// TIA Portal project "Paso a paso S7-1200 cambio giro bien en ambos sentidos intento completo final" (V16)

(* hardware
DEVICE "S7-1200 station_1"  S7-1200 Station
   slot 0: "Rack_0"  S7-1200 Rack  Rack  V1.0
   slot 1: "PLC_1"  CPU 1214C DC/DC/DC  6ES7 214-1AG31-0XB0  V3.0
*)

// ===== PLC "PLC_1"  CPU 1214C DC/DC/DC =====

VAR_GLOBAL   // PLC tag table "Tabla de variables estándar"
   "Marcha" AT %I0.1 : Bool;
   "Paro" AT %I0.2 : Bool;
   "IN1" AT %Q0.0 : Bool;
   "IN2" AT %Q0.1 : Bool;
   "IN3" AT %Q0.2 : Bool;
   "IN4" AT %Q0.3 : Bool;
   "marca_marcha" AT %M0.0 : Bool;
   "flanco_marcha" AT %M0.1 : Bool;
   "tiempo_trans" AT %MD2 : DInt;
   "marca_reinicio_temp" AT %M0.2 : Bool;
   "tiempo_actual" AT %MD6 : DInt;
   "marca1" AT %MD10 : Real;
   "marca2" AT %MD14 : Real;
   "Emergencia" AT %I0.3 : Bool;
   "Aumento" AT %I0.4 : Bool;
   "Freno" AT %I0.5 : Bool;
   "Conmutador cambio giro" AT %I0.6 : Bool;
   "flanco_aumento" AT %M0.3 : Bool;
   "flanco_freno" AT %M0.4 : Bool;
   "marca_bloqueo_aume_fre" AT %M0.5 : Bool;
   "flanco_paro" AT %M0.6 : Bool;
   "bloqueo_paro" AT %M0.7 : Bool;
   "marca3" AT %MD18 : Real;
   "tiempo_paro" AT %MW26 : Int;
   "marca_paro_a_0" AT %M1.0 : Bool;
   "marca_marcha2" AT %M1.1 : Bool;
   "flanco1" AT %M1.4 : Bool;
   "Inversor de giro" AT %I0.7 : Bool;
   "marca5" AT %M1.2 : Bool;
   "reinicio_counter" AT %M1.3 : Bool;
   "giro_izquierda" AT %M1.5 : Bool;
   "giro_derecha" AT %M1.6 : Bool;
   "estado_derecha" AT %M1.7 : Bool;
   "estado_izquierda" AT %M22.0 : Bool;
   "cambio a izq" AT %M22.1 : Bool;
   "tiempo_cambio" AT %MW30 : Int;
   "marca6" AT %M22.2 : Bool;
   "bloqueo_final" AT %M22.3 : Bool;
   "marca4" AT %MD32 : Real;
   "paro_bloqueo" AT %M22.4 : Bool;
   "tiempo para paro" AT %MW36 : Int;
END_VAR

// folder: System blocks/Program resources

DATA_BLOCK "IEC_Timer_0_DB"   // DB1
{ S7_Optimized_Access := 'TRUE' }
AUTHOR : Simatic
FAMILY : IEC
NAME : IEC_TMR
VERSION : 1.0
// stored: InstanceOfName IEC_TIMER
"IEC_TIMER"
BEGIN
END_DATA_BLOCK

DATA_BLOCK "IEC_Timer_0_DB_1"   // DB2
{ S7_Optimized_Access := 'TRUE' }
AUTHOR : Simatic
FAMILY : IEC
NAME : IEC_TMR
VERSION : 1.0
// stored: InstanceOfName IEC_TIMER
"IEC_TIMER"
BEGIN
END_DATA_BLOCK

DATA_BLOCK "IEC_Counter_0_DB"   // DB3
{ S7_Optimized_Access := 'TRUE' }
AUTHOR : Simatic
FAMILY : IEC
NAME : CNTR
VERSION : 1.0
// stored: InstanceOfName IEC_COUNTER
"IEC_COUNTER"
BEGIN
END_DATA_BLOCK

DATA_BLOCK "IEC_Timer_0_DB_2"   // DB4
{ S7_Optimized_Access := 'TRUE' }
AUTHOR : Simatic
FAMILY : IEC
NAME : IEC_TMR
VERSION : 1.0
// stored: InstanceOfName IEC_TIMER
"IEC_TIMER"
BEGIN
END_DATA_BLOCK

DATA_BLOCK "IEC_Counter_0_DB_1"   // DB5
{ S7_Optimized_Access := 'TRUE' }
AUTHOR : Simatic
FAMILY : IEC
NAME : CNTR
VERSION : 1.0
// stored: InstanceOfName IEC_COUNTER
"IEC_COUNTER"
BEGIN
END_DATA_BLOCK

DATA_BLOCK "IEC_Timer_0_DB_3"   // DB6
{ S7_Optimized_Access := 'TRUE' }
AUTHOR : Simatic
FAMILY : IEC
NAME : IEC_TMR
VERSION : 1.0
// stored: InstanceOfName IEC_TIMER
"IEC_TIMER"
BEGIN
END_DATA_BLOCK

// folder: (top level)

ORGANIZATION_BLOCK "Main"   // OB1, LAD, ProgramCycle
TITLE = "Main Program Sweep (Cycle)"
{ S7_Optimized_Access := 'TRUE' }
VERSION : 0.1
   VAR_TEMP   // added for the SCL form of the ladder/FBD networks
      _w1 : Bool;
      _w2 : Bool;
      _w3 : Bool;
      _w4 : Bool;
      _w5 : Bool;
   END_VAR
BEGIN

REGION Network 1: Marcha
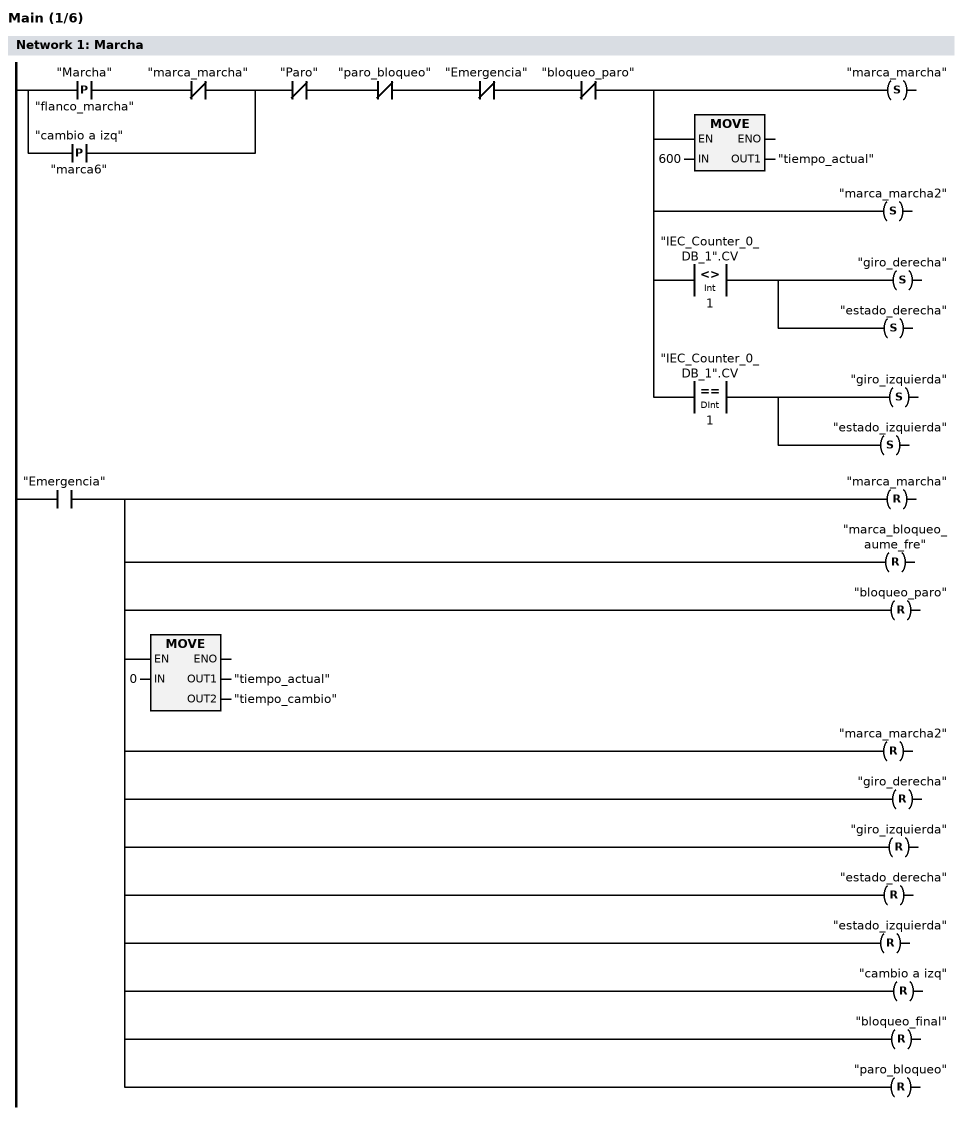
   RUNG wire#powerrail
      P_Contact(operand := "Marcha", bit := "flanco_marcha")
      I_Contact( "marca_marcha" )
      wire#w1
      I_Contact( "Paro" )
      I_Contact( "paro_bloqueo" )
      I_Contact( "Emergencia" )
      I_Contact( "bloqueo_paro" )
      wire#w2
      S_Coil( "marca_marcha" )
   END_RUNG
   RUNG wire#powerrail
      P_Contact(operand := "cambio a izq", bit := "marca6")
   END_RUNG wire#w1
   RUNG wire#w2
      { S7_GenerateENO := "TRUE" } Move(in := 600, out1 => "tiempo_actual")
   END_RUNG
   RUNG wire#w2
      S_Coil( "marca_marcha2" )
   END_RUNG
   RUNG wire#w2
      { S7_Templates := "SrcType := Int" } NE_Contact(in1 := "IEC_Counter_0_DB_1".CV, in2 := 1)
      wire#w3
      S_Coil( "giro_derecha" )
   END_RUNG
   RUNG wire#w3
      S_Coil( "estado_derecha" )
   END_RUNG
   RUNG wire#w2
      { S7_Templates := "SrcType := DInt" } EQ_Contact(in1 := "IEC_Counter_0_DB_1".CV, in2 := 1)
      wire#w4
      S_Coil( "giro_izquierda" )
   END_RUNG
   RUNG wire#w4
      S_Coil( "estado_izquierda" )
   END_RUNG
   RUNG wire#powerrail
      Contact( "Emergencia" )
      wire#w5
      R_Coil( "marca_marcha" )
   END_RUNG
   RUNG wire#w5
      R_Coil( "marca_bloqueo_aume_fre" )
   END_RUNG
   RUNG wire#w5
      R_Coil( "bloqueo_paro" )
   END_RUNG
   RUNG wire#w5
      { S7_GenerateENO := "TRUE" } Move(in := 0, out1 => "tiempo_actual", out2 => "tiempo_cambio")
   END_RUNG
   RUNG wire#w5
      R_Coil( "marca_marcha2" )
   END_RUNG
   RUNG wire#w5
      R_Coil( "giro_derecha" )
   END_RUNG
   RUNG wire#w5
      R_Coil( "giro_izquierda" )
   END_RUNG
   RUNG wire#w5
      R_Coil( "estado_derecha" )
   END_RUNG
   RUNG wire#w5
      R_Coil( "estado_izquierda" )
   END_RUNG
   RUNG wire#w5
      R_Coil( "cambio a izq" )
   END_RUNG
   RUNG wire#w5
      R_Coil( "bloqueo_final" )
   END_RUNG
   RUNG wire#w5
      R_Coil( "paro_bloqueo" )
   END_RUNG
   // the same network as SCL:
   #_w1 := "Marcha" AND NOT "flanco_marcha";   // rising edge of "Marcha"
   "flanco_marcha" := "Marcha";
   #_w2 := "cambio a izq" AND NOT "marca6";   // rising edge of "cambio a izq"
   "marca6" := "cambio a izq";
   #_w3 := ((#_w1 AND NOT "marca_marcha") OR #_w2) AND NOT "Paro" AND NOT "paro_bloqueo" AND NOT "Emergencia" AND NOT "bloqueo_paro";
   IF #_w3 THEN
       "marca_marcha" := TRUE;
       "tiempo_actual" := 600;
       "marca_marcha2" := TRUE;
   END_IF;
   IF #_w3 AND ("IEC_Counter_0_DB_1".CV <> 1) THEN
       "giro_derecha" := TRUE;
       "estado_derecha" := TRUE;
   END_IF;
   IF #_w3 AND ("IEC_Counter_0_DB_1".CV = 1) THEN
       "giro_izquierda" := TRUE;
       "estado_izquierda" := TRUE;
   END_IF;
   IF "Emergencia" THEN
       "marca_marcha" := FALSE;
       "marca_bloqueo_aume_fre" := FALSE;
       "bloqueo_paro" := FALSE;
       "tiempo_actual" := 0;
       "tiempo_cambio" := 0;
       "marca_marcha2" := FALSE;
       "giro_derecha" := FALSE;
       "giro_izquierda" := FALSE;
       "estado_derecha" := FALSE;
       "estado_izquierda" := FALSE;
       "cambio a izq" := FALSE;
       "bloqueo_final" := FALSE;
       "paro_bloqueo" := FALSE;
   END_IF;
END_REGION

REGION Network 2: Arranque progresivo
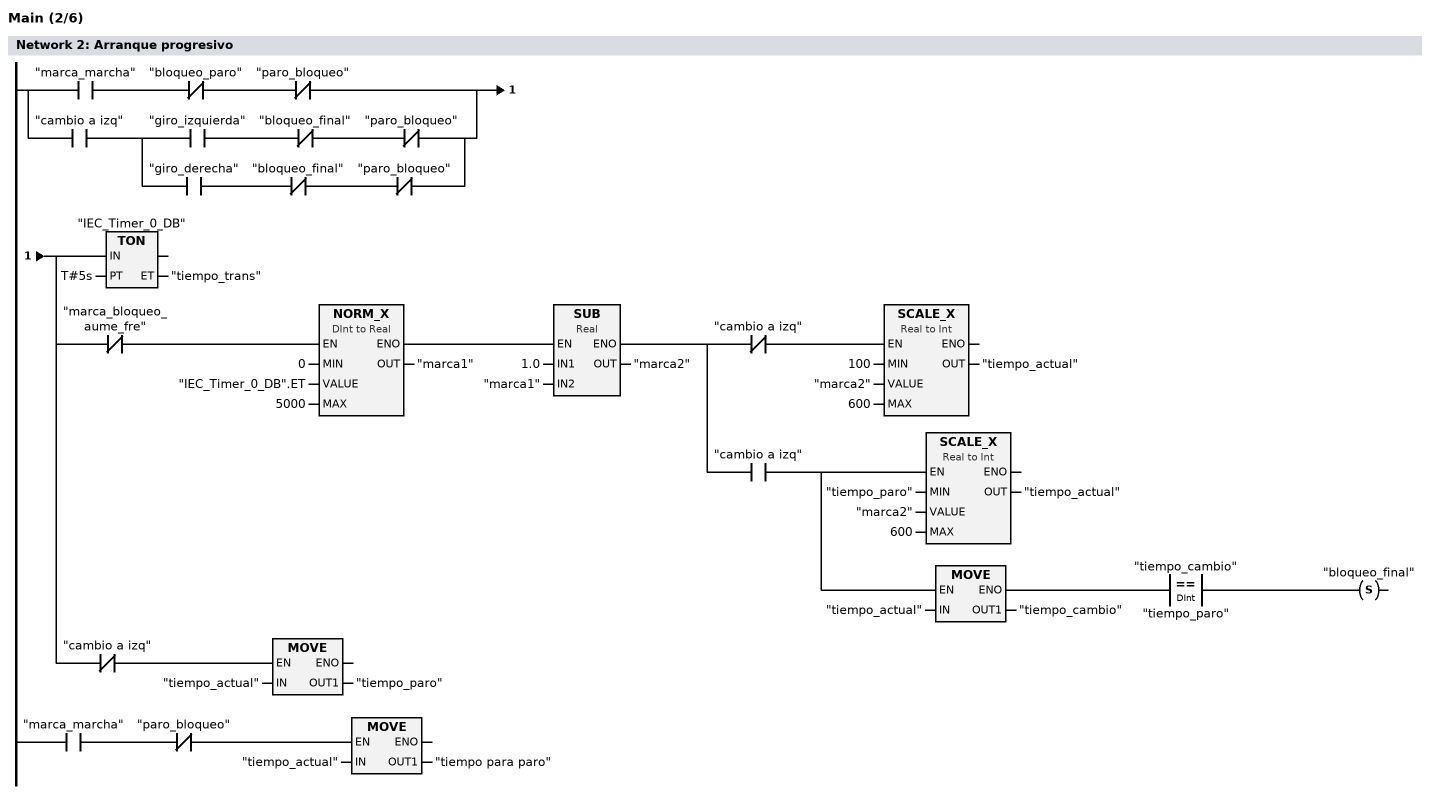
   // ENO of a box is taken as its EN; it also drops when the box reports an error
   #_w1 := ("marca_marcha" AND NOT "bloqueo_paro" AND NOT "paro_bloqueo") OR ("cambio a izq" AND (("giro_izquierda" AND NOT "bloqueo_final" AND NOT "paro_bloqueo") OR ("giro_derecha" AND NOT "bloqueo_final" AND NOT "paro_bloqueo")));
   "IEC_Timer_0_DB".TON(IN := #_w1, PT := T#5s, ET => "tiempo_trans");
   #_w2 := #_w1 AND NOT "marca_bloqueo_aume_fre";
   IF #_w2 THEN
       "marca1" := NORM_X(MIN := 0, VALUE := "IEC_Timer_0_DB".ET, MAX := 5000);
       "marca2" := 1.0 - "marca1";
   END_IF;
   IF #_w2 AND NOT "cambio a izq" THEN
       "tiempo_actual" := SCALE_X(MIN := 100, VALUE := "marca2", MAX := 600);
   END_IF;
   #_w3 := #_w2 AND "cambio a izq";
   IF #_w3 THEN
       "tiempo_actual" := SCALE_X(MIN := "tiempo_paro", VALUE := "marca2", MAX := 600);
       "tiempo_cambio" := "tiempo_actual";
   END_IF;
   IF #_w3 AND ("tiempo_cambio" = "tiempo_paro") THEN "bloqueo_final" := TRUE; END_IF;
   IF #_w1 AND NOT "cambio a izq" THEN "tiempo_paro" := "tiempo_actual"; END_IF;
   IF "marca_marcha" AND NOT "paro_bloqueo" THEN "tiempo para paro" := "tiempo_actual"; END_IF;
END_REGION

REGION Network 3: Secuencia salidas en ambos sentidos de giro
   // cambiar los contactor del conmutador de giro
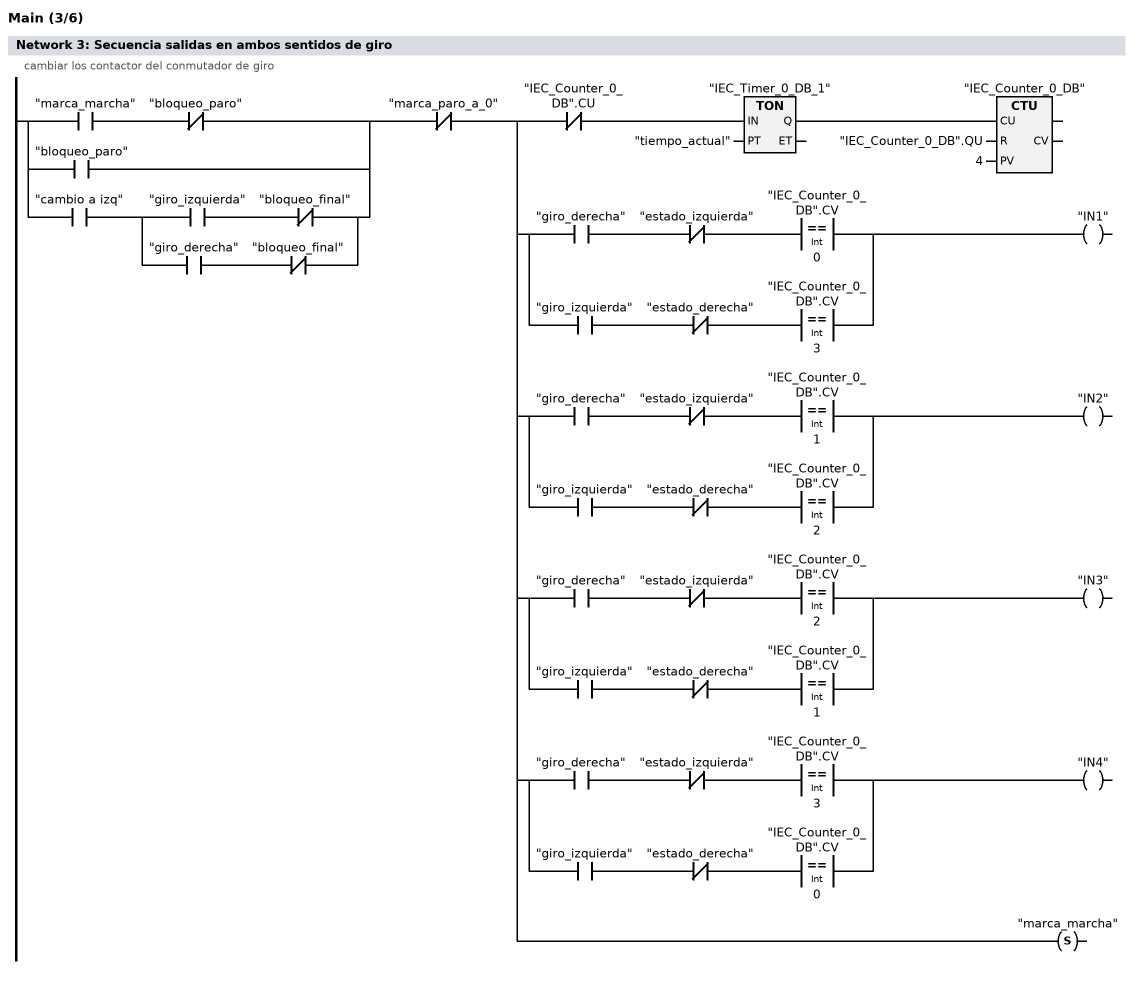
   #_w1 := (("marca_marcha" AND NOT "bloqueo_paro") OR "bloqueo_paro" OR ("cambio a izq" AND (("giro_izquierda" AND NOT "bloqueo_final") OR ("giro_derecha" AND NOT "bloqueo_final")))) AND NOT "marca_paro_a_0";
   "IEC_Timer_0_DB_1".TON(IN := #_w1 AND NOT "IEC_Counter_0_DB".CU, PT := "tiempo_actual");
   "IEC_Counter_0_DB".CTU(CU := "IEC_Timer_0_DB_1".Q, R := "IEC_Counter_0_DB".QU, PV := 4);
   "IN1" := #_w1 AND (("giro_derecha" AND NOT "estado_izquierda" AND ("IEC_Counter_0_DB".CV = 0)) OR ("giro_izquierda" AND NOT "estado_derecha" AND ("IEC_Counter_0_DB".CV = 3)));
   "IN2" := #_w1 AND (("giro_derecha" AND NOT "estado_izquierda" AND ("IEC_Counter_0_DB".CV = 1)) OR ("giro_izquierda" AND NOT "estado_derecha" AND ("IEC_Counter_0_DB".CV = 2)));
   "IN3" := #_w1 AND (("giro_derecha" AND NOT "estado_izquierda" AND ("IEC_Counter_0_DB".CV = 2)) OR ("giro_izquierda" AND NOT "estado_derecha" AND ("IEC_Counter_0_DB".CV = 1)));
   "IN4" := #_w1 AND (("giro_derecha" AND NOT "estado_izquierda" AND ("IEC_Counter_0_DB".CV = 3)) OR ("giro_izquierda" AND NOT "estado_derecha" AND ("IEC_Counter_0_DB".CV = 0)));
   IF #_w1 THEN "marca_marcha" := TRUE; END_IF;
END_REGION

REGION Network 4: Aumento y freno
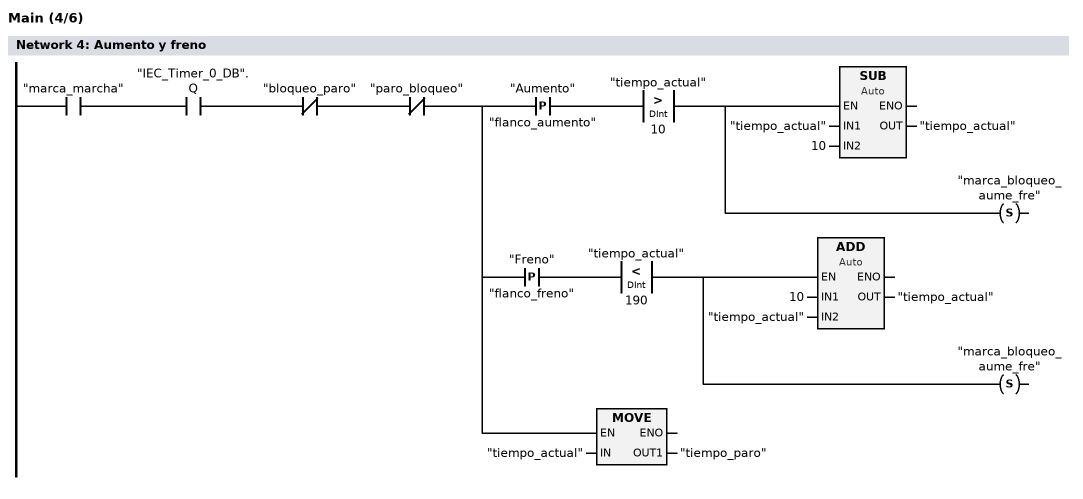
   RUNG wire#powerrail
      Contact( "marca_marcha" )
      Contact( "IEC_Timer_0_DB".Q )
      I_Contact( "bloqueo_paro" )
      I_Contact( "paro_bloqueo" )
      wire#w1
      P_Contact(operand := "Aumento", bit := "flanco_aumento")
      { S7_Templates := "SrcType := DInt" } GT_Contact(in1 := "tiempo_actual", in2 := 10)
      wire#w2
      { S7_GenerateENO := "TRUE" } Sub(in1 := "tiempo_actual", in2 := 10, out => "tiempo_actual")
   END_RUNG
   RUNG wire#w2
      S_Coil( "marca_bloqueo_aume_fre" )
   END_RUNG
   RUNG wire#w1
      P_Contact(operand := "Freno", bit := "flanco_freno")
      { S7_Templates := "SrcType := DInt" } LT_Contact(in1 := "tiempo_actual", in2 := 190)
      wire#w3
      { S7_GenerateENO := "TRUE" } Add(in1 := 10, in2 := "tiempo_actual", out => "tiempo_actual")
   END_RUNG
   RUNG wire#w3
      S_Coil( "marca_bloqueo_aume_fre" )
   END_RUNG
   RUNG wire#w1
      { S7_GenerateENO := "TRUE" } Move(in := "tiempo_actual", out1 => "tiempo_paro")
   END_RUNG
   // the same network as SCL:
   #_w1 := "marca_marcha" AND "IEC_Timer_0_DB".Q AND NOT "bloqueo_paro" AND NOT "paro_bloqueo";
   #_w2 := #_w1 AND "Aumento" AND NOT "flanco_aumento";   // rising edge of "Aumento"
   "flanco_aumento" := "Aumento";
   #_w3 := #_w2 AND ("tiempo_actual" > 10);
   IF #_w3 THEN
       "tiempo_actual" := "tiempo_actual" - 10;
       "marca_bloqueo_aume_fre" := TRUE;
   END_IF;
   #_w4 := #_w1 AND "Freno" AND NOT "flanco_freno";   // rising edge of "Freno"
   "flanco_freno" := "Freno";
   #_w5 := #_w4 AND ("tiempo_actual" < 190);
   IF #_w5 THEN
       "tiempo_actual" := 10 + "tiempo_actual";
       "marca_bloqueo_aume_fre" := TRUE;
   END_IF;
   IF #_w1 THEN "tiempo_paro" := "tiempo_actual"; END_IF;
END_REGION

REGION Network 5: Cambio de giro
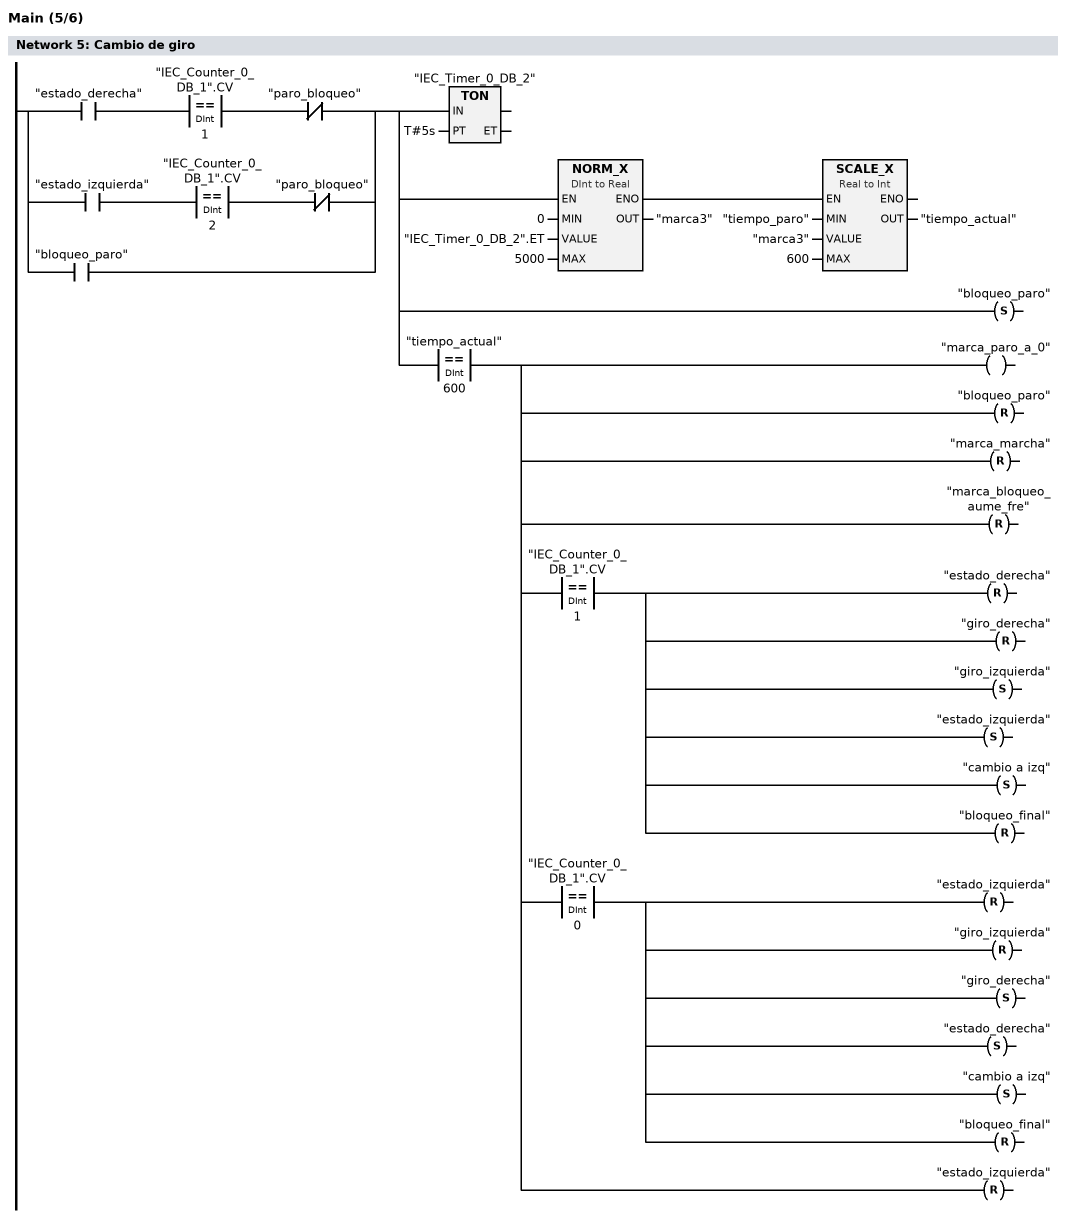
   // ENO of a box is taken as its EN; it also drops when the box reports an error
   #_w1 := ("estado_derecha" AND ("IEC_Counter_0_DB_1".CV = 1) AND NOT "paro_bloqueo") OR ("estado_izquierda" AND ("IEC_Counter_0_DB_1".CV = 2) AND NOT "paro_bloqueo") OR "bloqueo_paro";
   "IEC_Timer_0_DB_2".TON(IN := #_w1, PT := T#5s);
   IF #_w1 THEN
       "marca3" := NORM_X(MIN := 0, VALUE := "IEC_Timer_0_DB_2".ET, MAX := 5000);
       "tiempo_actual" := SCALE_X(MIN := "tiempo_paro", VALUE := "marca3", MAX := 600);
       "bloqueo_paro" := TRUE;
   END_IF;
   "marca_paro_a_0" := #_w1 AND ("tiempo_actual" = 600);
   IF "marca_paro_a_0" THEN
       "bloqueo_paro" := FALSE;
       "marca_marcha" := FALSE;
       "marca_bloqueo_aume_fre" := FALSE;
   END_IF;
   IF "marca_paro_a_0" AND ("IEC_Counter_0_DB_1".CV = 1) THEN
       "estado_derecha" := FALSE;
       "giro_derecha" := FALSE;
       "giro_izquierda" := TRUE;
       "estado_izquierda" := TRUE;
       "cambio a izq" := TRUE;
       "bloqueo_final" := FALSE;
   END_IF;
   IF "marca_paro_a_0" AND ("IEC_Counter_0_DB_1".CV = 0) THEN
       "estado_izquierda" := FALSE;
       "giro_izquierda" := FALSE;
       "giro_derecha" := TRUE;
       "estado_derecha" := TRUE;
       "cambio a izq" := TRUE;
       "bloqueo_final" := FALSE;
   END_IF;
   IF "marca_paro_a_0" THEN "estado_izquierda" := FALSE; END_IF;
END_REGION

REGION Network 6: Paro
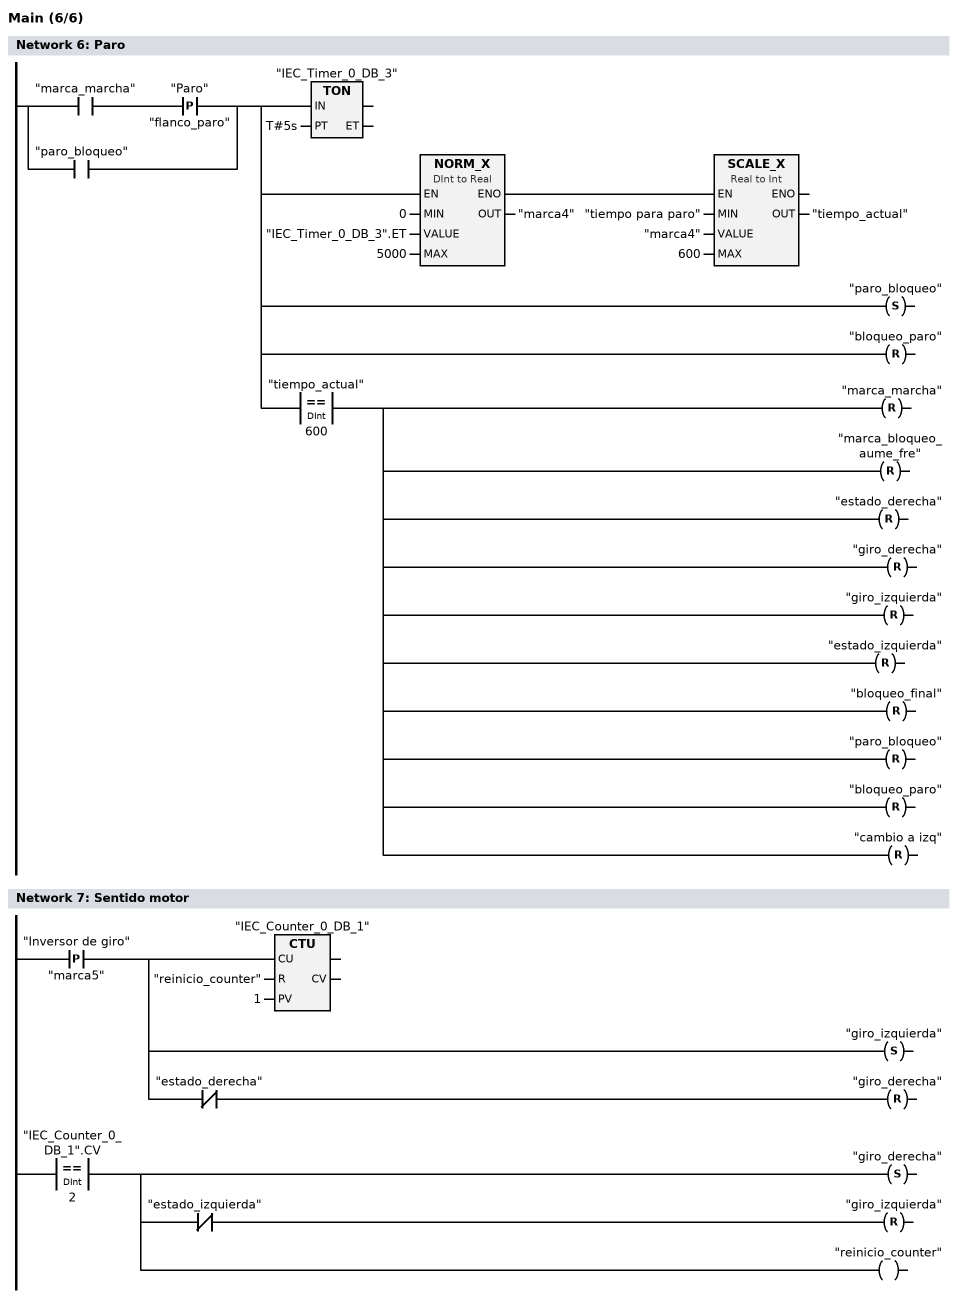
   // ENO of a box is taken as its EN; it also drops when the box reports an error
   #_w1 := "marca_marcha" AND "Paro" AND NOT "flanco_paro";   // rising edge of "Paro"
   "flanco_paro" := "Paro";
   #_w2 := #_w1 OR "paro_bloqueo";
   "IEC_Timer_0_DB_3".TON(IN := #_w2, PT := T#5s);
   IF #_w2 THEN
       "marca4" := NORM_X(MIN := 0, VALUE := "IEC_Timer_0_DB_3".ET, MAX := 5000);
       "tiempo_actual" := SCALE_X(MIN := "tiempo para paro", VALUE := "marca4", MAX := 600);
       "paro_bloqueo" := TRUE;
       "bloqueo_paro" := FALSE;
   END_IF;
   IF #_w2 AND ("tiempo_actual" = 600) THEN
       "marca_marcha" := FALSE;
       "marca_bloqueo_aume_fre" := FALSE;
       "estado_derecha" := FALSE;
       "giro_derecha" := FALSE;
       "giro_izquierda" := FALSE;
       "estado_izquierda" := FALSE;
       "bloqueo_final" := FALSE;
       "paro_bloqueo" := FALSE;
       "bloqueo_paro" := FALSE;
       "cambio a izq" := FALSE;
   END_IF;
END_REGION

REGION Network 7: Sentido motor
   #_w1 := "Inversor de giro" AND NOT "marca5";   // rising edge of "Inversor de giro"
   "marca5" := "Inversor de giro";
   "IEC_Counter_0_DB_1".CTU(CU := #_w1, R := "reinicio_counter", PV := 1);
   IF #_w1 THEN "giro_izquierda" := TRUE; END_IF;
   IF #_w1 AND NOT "estado_derecha" THEN "giro_derecha" := FALSE; END_IF;
   #_w2 := "IEC_Counter_0_DB_1".CV = 2;
   IF #_w2 THEN "giro_derecha" := TRUE; END_IF;
   IF #_w2 AND NOT "estado_izquierda" THEN "giro_izquierda" := FALSE; END_IF;
   "reinicio_counter" := #_w2;
END_REGION
END_ORGANIZATION_BLOCK